FUNCTION_BLOCK UnitControl
  (* Standard: 61499-2 *)
  (* Version 0.1, 2014-00-16, Canto-Air, CANTO-AIR-PC *)
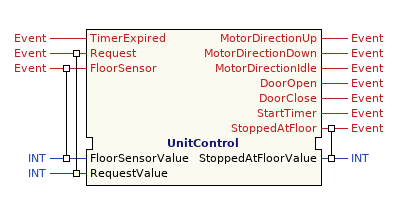
  EVENT_INPUT
    TimerExpired;
    Request WITH RequestValue;
    FloorSensor WITH FloorSensorValue;
  END_EVENT
  EVENT_OUTPUT
    MotorDirectionUp;
    MotorDirectionDown;
    MotorDirectionIdle;
    DoorOpen;
    DoorClose;
    StartTimer;
    StoppedAtFloor WITH StoppedAtFloorValue;
  END_EVENT
  VAR_INPUT
    FloorSensorValue : INT;
    RequestValue : INT;
  END_VAR
  VAR_OUTPUT
    StoppedAtFloorValue : INT;
  END_VAR
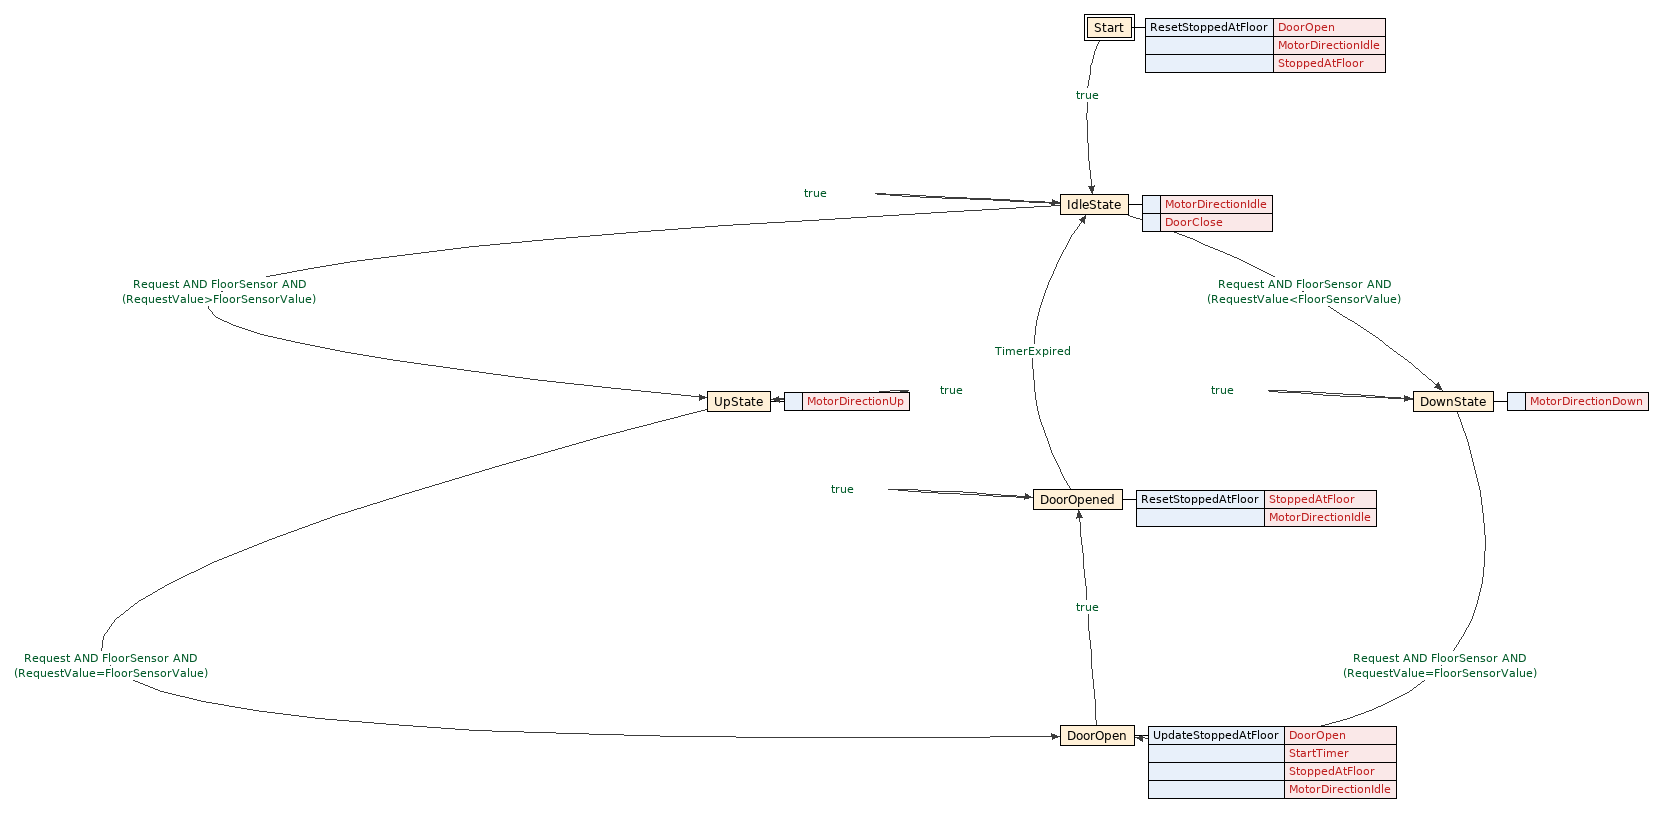
  EC_STATES
    Start : ResetStoppedAtFloor -> DoorOpen, -> MotorDirectionIdle, -> StoppedAtFloor;
    IdleState : -> MotorDirectionIdle, -> DoorClose;
    UpState : -> MotorDirectionUp;
    DoorOpen : UpdateStoppedAtFloor -> DoorOpen, -> StartTimer, -> StoppedAtFloor, -> MotorDirectionIdle;
    DownState : -> MotorDirectionDown;
    DoorOpened : ResetStoppedAtFloor -> StoppedAtFloor, -> MotorDirectionIdle;
  END_STATES
  EC_TRANSITIONS
    Start TO IdleState := true;
    IdleState TO UpState := Request AND FloorSensor AND (RequestValue>FloorSensorValue);
    IdleState TO DownState := Request AND FloorSensor AND (RequestValue<FloorSensorValue);
    IdleState TO IdleState := true;
    UpState TO DoorOpen := Request AND FloorSensor AND (RequestValue=FloorSensorValue);
    UpState TO UpState := true;
    DoorOpen TO DoorOpened := true;
    DownState TO DoorOpen := Request AND FloorSensor AND (RequestValue=FloorSensorValue);
    DownState TO DownState := true;
    DoorOpened TO IdleState := TimerExpired;
    DoorOpened TO DoorOpened := true;
  END_TRANSITIONS
  ALGORITHM UpdateStoppedAtFloor IN C:
me->StoppedAtFloorValue =  me->FloorSensorValue;
  END_ALGORITHM
  ALGORITHM ResetStoppedAtFloor IN C:
me->StoppedAtFloorValue =  -1;
  END_ALGORITHM
END_FUNCTION_BLOCK
